VISUALIZATION NavBarEmpty_1  // 200x880
END_VISUALIZATION

(* stored: Version 1.1.0.1, ProductVersion 3.1.4024.12
   Visu NavBarEmpty_1: Id {3acce945-5cd8-4a57-977c-ccf93230bf1d} *)
